TYPE T_BCH_ID :
STRUCT
	Bch: INT;
	Bch_Bcc: INT;
	Bch_Bcc_Bcd: INT;
END_STRUCT
END_TYPE

(* stored: Version 1.1.0.1, ProductVersion 3.1.0.26
   DUT T_BCH_ID: Id {4c3c8207-4514-47ab-82e4-c7142d181686} *)
